(* IEC 61131-3 sources: com.logicals.lc3.webinar/usRTS_RPMControl_iSOC/src_FB_LIB_SAFE/Numeric/ULINT, 8 files *)

(* ---- wADD_ULINT_2.iecst ---- *)
NAMESPACE logicals.web.standard
NAMESPACE numeric

/*
 * Function block wrapper for IEC 61131-3 ADD<br>
 * IN1 =  1st value (ULINT)<br>
 * IN2 =  2nd value (ULINT)<br>
 * OUT = Sum of all input values (ULINT)<br>
 */
FUNCTION_BLOCK wADD_ULINT_2
	{ vNameAlignment:="center"; altName:="+"; bgColor:="Plum"; width:=40; hideIONames; }
	VAR_INPUT
		IN1 : ULINT;
		IN2 : ULINT;
	END_VAR
	VAR_OUTPUT
		OUT : ULINT;
	END_VAR

	OUT := ADD(IN1:=IN1, IN2:=IN2, ENO=>ENO);
END_FUNCTION_BLOCK

END_NAMESPACE
END_NAMESPACE

(* ---- wADD_ULINT_3.iecst ---- *)
NAMESPACE logicals.web.standard
NAMESPACE numeric

/*
 * Function block wrapper for IEC 61131-3 ADD<br>
 * IN1 =  1st value (ULINT)<br>
 * IN2 =  2nd value (ULINT)<br>
 * IN3 =  3rd value (ULINT)<br>
 * OUT = Sum of all input values (ULINT)<br>
 */
FUNCTION_BLOCK wADD_ULINT_3
	{ vNameAlignment:="center"; altName:="+"; bgColor:="Plum"; width:=40; hideIONames; }
	VAR_INPUT
		IN1 : ULINT;
		IN2 : ULINT;
		IN3 : ULINT;
	END_VAR
	VAR_OUTPUT
		OUT : ULINT;
	END_VAR

	OUT := ADD(IN1:=IN1, IN2:=IN2, IN3:=IN3, ENO=>ENO);
END_FUNCTION_BLOCK

END_NAMESPACE
END_NAMESPACE

(* ---- wADD_ULINT_4.iecst ---- *)
NAMESPACE logicals.web.standard
NAMESPACE numeric

/*
 * Function block wrapper for IEC 61131-3 ADD<br>
 * IN1 =  1st value (ULINT)<br>
 * IN2 =  2nd value (ULINT)<br>
 * IN3 =  3rd value (ULINT)<br>
 * IN4 =  4th value (ULINT)<br>
 * OUT = Sum of all input values (ULINT)<br>
 */
FUNCTION_BLOCK wADD_ULINT_4
	{ vNameAlignment:="center"; altName:="+"; bgColor:="Plum"; width:=40; hideIONames; }
	VAR_INPUT
		IN1 : ULINT;
		IN2 : ULINT;
		IN3 : ULINT;
		IN4 : ULINT;
	END_VAR
	VAR_OUTPUT
		OUT : ULINT;
	END_VAR

	OUT := ADD(IN1:=IN1, IN2:=IN2, IN3:=IN3, IN4:=IN4, ENO=>ENO);
END_FUNCTION_BLOCK

END_NAMESPACE
END_NAMESPACE

(* ---- wDIV_ULINT.iecst ---- *)
NAMESPACE logicals.web.standard
NAMESPACE numeric

/*
 * Function block wrapper for IEC 61131-3 DIV<br>
 * IN1 =  1st value (ULINT)<br>
 * IN2 =  2nd value (ULINT)<br>
 * OUT = quotient of IN1 divided by IN2 (ULINT)<br>
 */
FUNCTION_BLOCK wDIV_ULINT
	{ vNameAlignment:="center"; altName:="/"; bgColor:="Plum"; width:=40; hideIONames; }
	VAR_INPUT
		IN1 : ULINT;
		IN2 : ULINT;
	END_VAR
	VAR_OUTPUT
		OUT : ULINT;
	END_VAR

	OUT := DIV(IN1:=IN1, IN2:=IN2, ENO=>ENO);
END_FUNCTION_BLOCK

END_NAMESPACE
END_NAMESPACE

(* ---- wMUL_ULINT_2.iecst ---- *)
NAMESPACE logicals.web.standard
NAMESPACE numeric

/*
 * Function block wrapper for IEC 61131-3 MUL<br>
 * IN1 =  1st value (ULINT)<br>
 * IN2 =  2nd value (ULINT)<br>
 * OUT = Product of multiplication of all inputs (ULINT)<br>
 */
FUNCTION_BLOCK wMUL_ULINT_2
	{ vNameAlignment:="center"; altName:="*"; bgColor:="Plum"; width:=40; hideIONames; }
	VAR_INPUT
		IN1 : ULINT;
		IN2 : ULINT;
	END_VAR
	VAR_OUTPUT
		OUT : ULINT;
	END_VAR

	OUT := MUL(IN1:=IN1, IN2:=IN2, ENO=>ENO);
END_FUNCTION_BLOCK

END_NAMESPACE
END_NAMESPACE

(* ---- wMUL_ULINT_3.iecst ---- *)
NAMESPACE logicals.web.standard
NAMESPACE numeric

/*
 * Function block wrapper for IEC 61131-3 MUL<br>
 * IN1 =  1st value (ULINT)<br>
 * IN2 =  2nd value (ULINT)<br>
 * IN3 =  3rd value (ULINT)<br>
 * OUT = Product of multiplication of all inputs (ULINT)<br>
 */
FUNCTION_BLOCK wMUL_ULINT_3
	{ vNameAlignment:="center"; altName:="*"; bgColor:="Plum"; width:=40; hideIONames; }
	VAR_INPUT
		IN1 : ULINT;
		IN2 : ULINT;
		IN3 : ULINT;
	END_VAR
	VAR_OUTPUT
		OUT : ULINT;
	END_VAR

	OUT := MUL(IN1:=IN1, IN2:=IN2, IN3:=IN3, ENO=>ENO);
END_FUNCTION_BLOCK

END_NAMESPACE
END_NAMESPACE

(* ---- wMUL_ULINT_4.iecst ---- *)
NAMESPACE logicals.web.standard
NAMESPACE numeric

/*
 * Function block wrapper for IEC 61131-3 MUL<br>
 * IN1 =  1st value (ULINT)<br>
 * IN2 =  2nd value (ULINT)<br>
 * IN3 =  3rd value (ULINT)<br>
 * IN4 =  4th value (ULINT)<br>
 * OUT = Product of multiplication of all inputs (ULINT)<br>
 */
FUNCTION_BLOCK wMUL_ULINT_4
	{ vNameAlignment:="center"; altName:="*"; bgColor:="Plum"; width:=40; hideIONames; }
	VAR_INPUT
		IN1 : ULINT;
		IN2 : ULINT;
		IN3 : ULINT;
		IN4 : ULINT;
	END_VAR
	VAR_OUTPUT
		OUT : ULINT;
	END_VAR

	OUT := MUL(IN1:=IN1, IN2:=IN2, IN3:=IN3, IN4:=IN4, ENO=>ENO);
END_FUNCTION_BLOCK

END_NAMESPACE
END_NAMESPACE

(* ---- wSUB_ULINT.iecst ---- *)
NAMESPACE logicals.web.standard
NAMESPACE numeric

/*
 * Function block wrapper for IEC 61131-3 SUB<br>
 * IN1 =  1st value (ULINT)<br>
 * IN2 =  2nd value (ULINT)<br>
 * OUT = IN1 minus IN2 (ULINT)<br>
 */
FUNCTION_BLOCK wSUB_ULINT
	{ vNameAlignment:="center"; altName:="-"; bgColor:="Plum"; width:=40; hideIONames; }
	VAR_INPUT
		IN1 : ULINT;
		IN2 : ULINT;
	END_VAR
	VAR_OUTPUT
		OUT : ULINT;
	END_VAR

	OUT := SUB(IN1:=IN1, IN2:=IN2, ENO=>ENO);
END_FUNCTION_BLOCK

END_NAMESPACE
END_NAMESPACE
